// TIA Portal V18 export
TYPE "RCS_SysCount_V1"
// stored: IsFailsafeCompliant false
   STRUCT
      OK : Array[0..14] of DInt;   // [0]Total Count
      NG : Array[0..14] of DInt;   // [0]Total Count
      Total : DInt;
      OKHolding : DInt;
      NGHolding : DInt;
      TotalHolding : DInt;
      ClearOK : Bool;
      ClearNG : Bool;
      ClearTotal : Bool;
   END_STRUCT;
END_TYPE
